# EPICS IOC start-up script: iocsh/ethercatmcBinaryOutReadback.iocsh
ethercatmcCreateAsynParam $(MOTOR_PORT) $(ASYNPARAMNAME) Int32

dbLoadRecords("ethercatmcBinaryOutReadback.template", "P=$(P), R=$(R), MOTOR_PORT=$(MOTOR_PORT), CHNO=$(CHNO), ASYNPARAMNAME=$(ASYNPARAMNAME), DESC=$(DESC), ZNAM=$(ZNAM), ONAM=$(ONAM)")
